PROGRAM Test
VAR
END_VAR

IF TRUE THEN
	Act_Test();
END_IF

ACTION Act_Test:
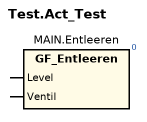
MAIN.Entleeren(); // GF_Entleeren
END_ACTION

END_PROGRAM

(* stored: Version 1.1.0.1, ProductVersion 3.1.4024.12
   POU Test: Id {f9be35fc-e271-4a1f-9fd1-0dae8763ecd1}, SpecialFunc None
   Action Act_Test: Id {b6a48476-98a7-4aca-953b-bf0fedc6c393} *)
